% RSLogix 500 project Blue Banner Dump Line SLC 500.RSS, saved by version 11.00.00.00 %
PROJECT "BLUEBANR"    % processor: type code 8 %

PROGRAM FILES
  LAD 2   56 rungs

DATA FILES
  O0 OUTPUT  2 elements
  I1 INPUT  3 elements
  S2 STATUS  16 elements
  B3 BINARY  3 elements
  T4 TIMER  18 elements
  C5 COUNTER  1 elements
  R6 CONTROL  1 elements
  N7 INTEGER  1 elements

LADDER 2
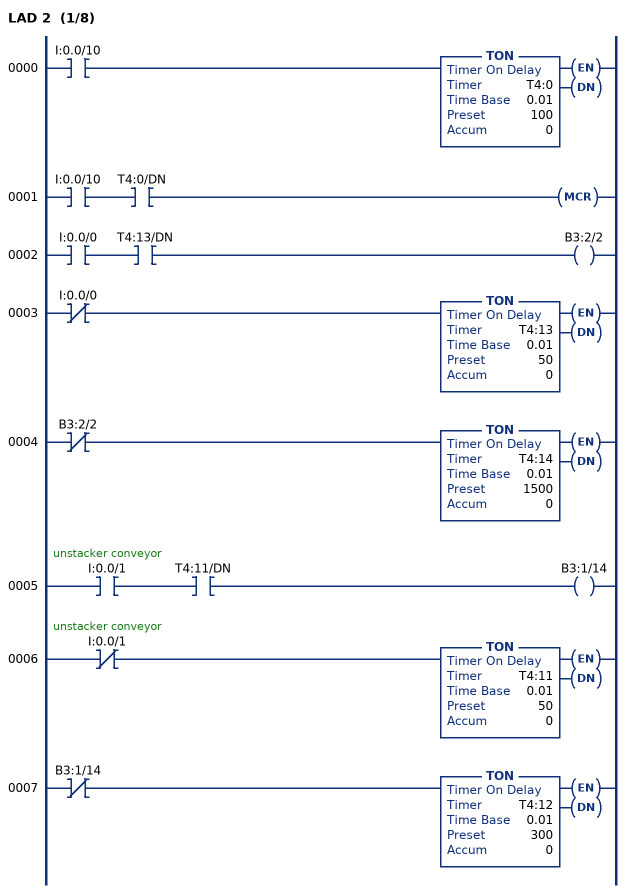
% Rung: 0 %
SOR XIC I:0.0/10 TON T4:0 0.01 100 0 EOR
% Rung: 1 %
SOR XIC I:0.0/10 XIC T4:0/DN MCR EOR
% Rung: 2 %
SOR XIC I:0.0/0 XIC T4:13/DN OTE B3:2/2 EOR
% Rung: 3 %
SOR XIO I:0.0/0 TON T4:13 0.01 50 0 EOR
% Rung: 4 %
SOR XIO B3:2/2 TON T4:14 0.01 1500 0 EOR
% Rung: 5 %
SOR XIC I:0.0/1 XIC T4:11/DN OTE B3:1/14 EOR
%   I:0.0/1  "unstacker conveyor" %
% Rung: 6 %
SOR XIO I:0.0/1 TON T4:11 0.01 50 0 EOR
%   I:0.0/1  "unstacker conveyor" %
% Rung: 7 %
SOR XIO B3:1/14 TON T4:12 0.01 300 0 EOR

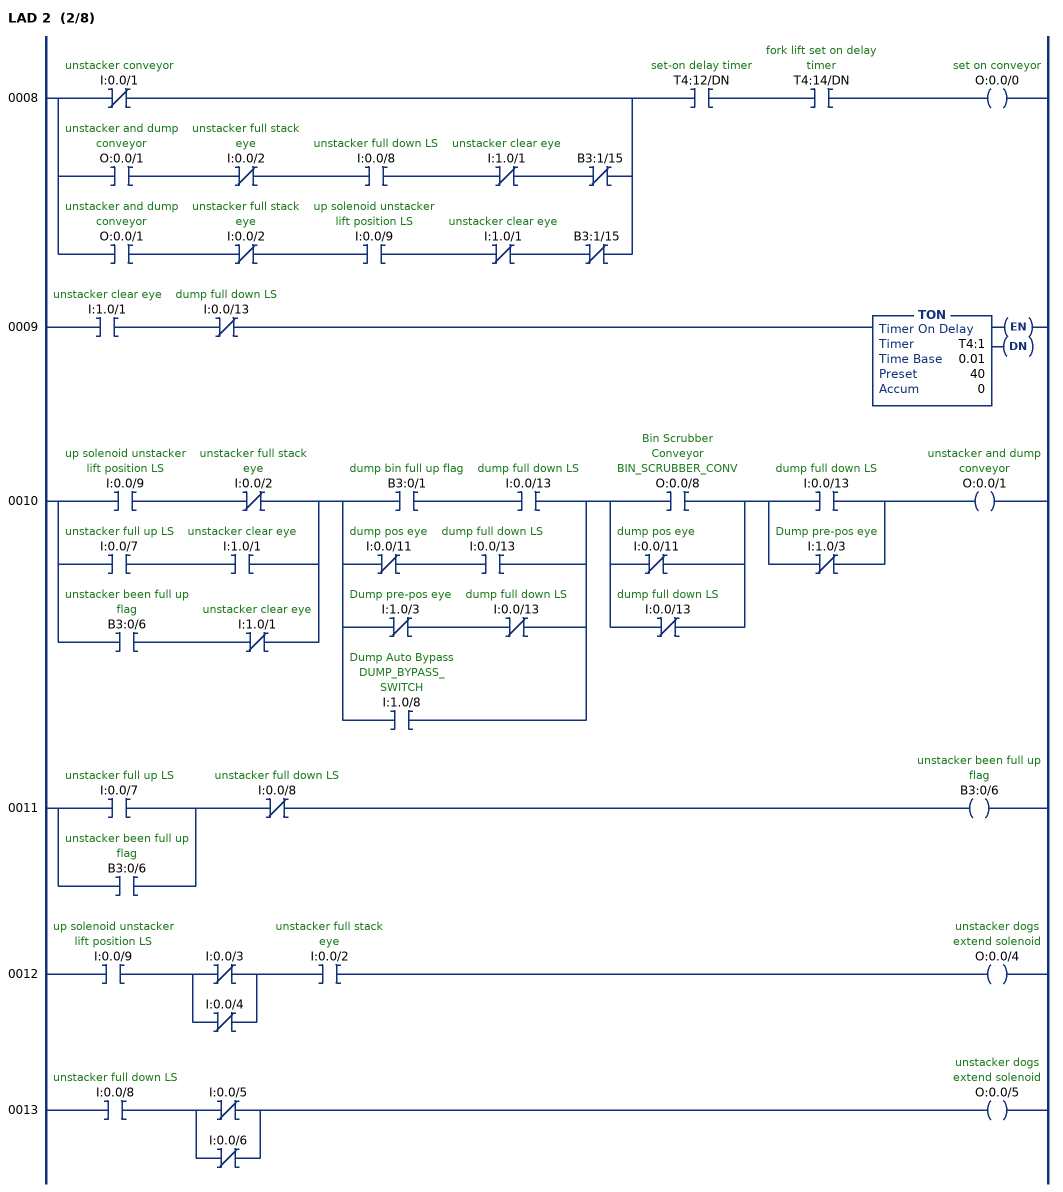
% Rung: 8 %
SOR BST XIO I:0.0/1 NXB XIC O:0.0/1 XIO I:0.0/2 XIC I:0.0/8 XIO I:1.0/1 XIO B3:1/15 NXB XIC O:0.0/1 XIO I:0.0/2 XIC I:0.0/9 XIO I:1.0/1 XIO B3:1/15 BND XIC T4:12/DN XIC T4:14/DN OTE O:0.0/0 EOR
%   I:0.0/1  "unstacker conveyor" %
%   O:0.0/1  "unstacker and dump conveyor" %
%   I:0.0/2  "unstacker full stack eye" %
%   I:0.0/8  "unstacker full down LS" %
%   I:1.0/1  "unstacker clear eye" %
%   I:0.0/9  "up solenoid unstacker lift position LS" %
%   T4:12/DN  "set-on delay timer" %
%   T4:14/DN  "fork lift set on delay timer" %
%   O:0.0/0  "set on conveyor" %
% Rung: 9 %
SOR XIC I:1.0/1 XIO I:0.0/13 TON T4:1 0.01 40 0 EOR
%   I:1.0/1  "unstacker clear eye" %
%   I:0.0/13  "dump full down LS" %
% Rung: 10 %
SOR BST XIC I:0.0/9 XIO I:0.0/2 NXB XIC I:0.0/7 XIC I:1.0/1 NXB XIC B3:0/6 XIO I:1.0/1 BND BST XIC B3:0/1 XIC I:0.0/13 NXB XIO I:0.0/11 XIC I:0.0/13 NXB BST XIO I:1.0/3 XIO I:0.0/13 NXB XIC I:1.0/8 BND BND BST XIC O:0.0/8 NXB XIO I:0.0/11 NXB XIO I:0.0/13 BND BST XIC I:0.0/13 NXB XIO I:1.0/3 BND OTE O:0.0/1 EOR
%   I:0.0/9  "up solenoid unstacker lift position LS" %
%   I:0.0/2  "unstacker full stack eye" %
%   I:0.0/7  "unstacker full up LS" %
%   I:1.0/1  "unstacker clear eye" %
%   B3:0/6  "unstacker been full up flag" %
%   B3:0/1  "dump bin full up flag" %
%   I:0.0/13  "dump full down LS" %
%   I:0.0/11  "dump pos eye" %
%   I:1.0/3  "Dump pre-pos eye" %
%   I:1.0/8  DUMP_BYPASS_SWITCH  "Dump Auto Bypass" %
%   O:0.0/8  BIN_SCRUBBER_CONV  "Bin Scrubber Conveyor" %
%   O:0.0/1  "unstacker and dump conveyor" %
% Rung: 11 %
SOR BST XIC I:0.0/7 NXB XIC B3:0/6 BND XIO I:0.0/8 OTE B3:0/6 EOR
%   I:0.0/7  "unstacker full up LS" %
%   B3:0/6  "unstacker been full up flag" %
%   I:0.0/8  "unstacker full down LS" %
% Rung: 12 %
SOR XIC I:0.0/9 BST XIO I:0.0/3 NXB XIO I:0.0/4 BND XIC I:0.0/2 OTE O:0.0/4 EOR
%   I:0.0/9  "up solenoid unstacker lift position LS" %
%   I:0.0/2  "unstacker full stack eye" %
%   O:0.0/4  "unstacker dogs extend solenoid" %
% Rung: 13 %
SOR XIC I:0.0/8 BST XIO I:0.0/5 NXB XIO I:0.0/6 BND OTE O:0.0/5 EOR
%   I:0.0/8  "unstacker full down LS" %
%   O:0.0/5  "unstacker dogs extend solenoid" %

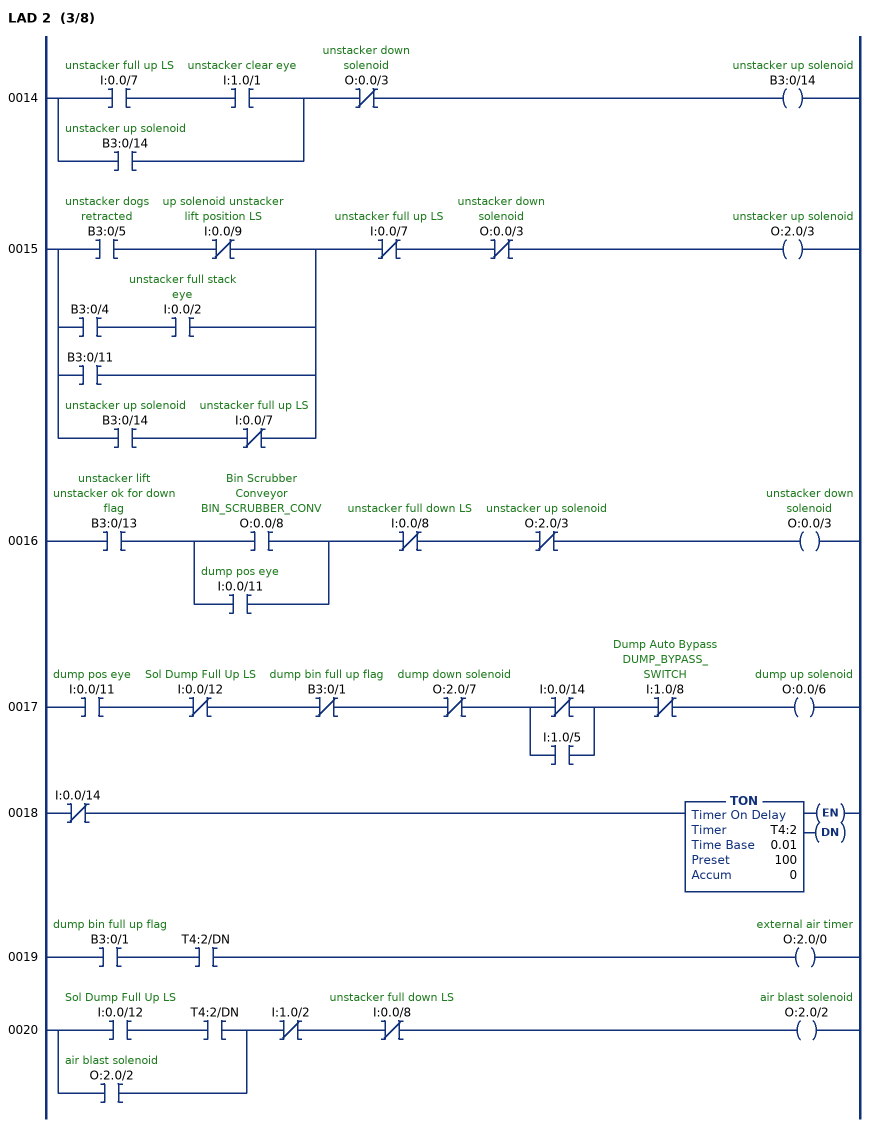
% Rung: 14 %
SOR BST XIC I:0.0/7 XIC I:1.0/1 NXB XIC B3:0/14 BND XIO O:0.0/3 OTE B3:0/14 EOR
%   I:0.0/7  "unstacker full up LS" %
%   I:1.0/1  "unstacker clear eye" %
%   B3:0/14  "unstacker up solenoid" %
%   O:0.0/3  "unstacker down solenoid" %
% Rung: 15 %
SOR BST XIC B3:0/5 XIO I:0.0/9 NXB XIC B3:0/4 XIC I:0.0/2 NXB XIC B3:0/11 NXB XIC B3:0/14 XIO I:0.0/7 BND XIO I:0.0/7 XIO O:0.0/3 OTE O:2.0/3 EOR
%   B3:0/5  "unstacker dogs retracted" %
%   I:0.0/9  "up solenoid unstacker lift position LS" %
%   I:0.0/2  "unstacker full stack eye" %
%   B3:0/14  "unstacker up solenoid" %
%   I:0.0/7  "unstacker full up LS" %
%   O:0.0/3  "unstacker down solenoid" %
%   O:2.0/3  "unstacker up solenoid" %
% Rung: 16 %
SOR XIC B3:0/13 BST XIC O:0.0/8 NXB XIC I:0.0/11 BND XIO I:0.0/8 XIO O:2.0/3 OTE O:0.0/3 EOR
%   B3:0/13  "unstacker lift unstacker ok for down flag" %
%   O:0.0/8  BIN_SCRUBBER_CONV  "Bin Scrubber Conveyor" %
%   I:0.0/11  "dump pos eye" %
%   I:0.0/8  "unstacker full down LS" %
%   O:2.0/3  "unstacker up solenoid" %
%   O:0.0/3  "unstacker down solenoid" %
% Rung: 17 %
SOR XIC I:0.0/11 XIO I:0.0/12 XIO B3:0/1 XIO O:2.0/7 BST XIO I:0.0/14 NXB XIC I:1.0/5 BND XIO I:1.0/8 OTE O:0.0/6 EOR
%   I:0.0/11  "dump pos eye" %
%   I:0.0/12  "Sol Dump Full Up LS" %
%   B3:0/1  "dump bin full up flag" %
%   O:2.0/7  "dump down solenoid" %
%   I:1.0/8  DUMP_BYPASS_SWITCH  "Dump Auto Bypass" %
%   O:0.0/6  "dump up solenoid" %
% Rung: 18 %
SOR XIO I:0.0/14 TON T4:2 0.01 100 0 EOR
% Rung: 19 %
SOR XIC B3:0/1 XIC T4:2/DN OTE O:2.0/0 EOR
%   B3:0/1  "dump bin full up flag" %
%   O:2.0/0  "external air timer" %
% Rung: 20 %
SOR BST XIC I:0.0/12 XIC T4:2/DN NXB XIC O:2.0/2 BND XIO I:1.0/2 XIO I:0.0/8 OTE O:2.0/2 EOR
%   I:0.0/12  "Sol Dump Full Up LS" %
%   O:2.0/2  "air blast solenoid" %
%   I:0.0/8  "unstacker full down LS" %

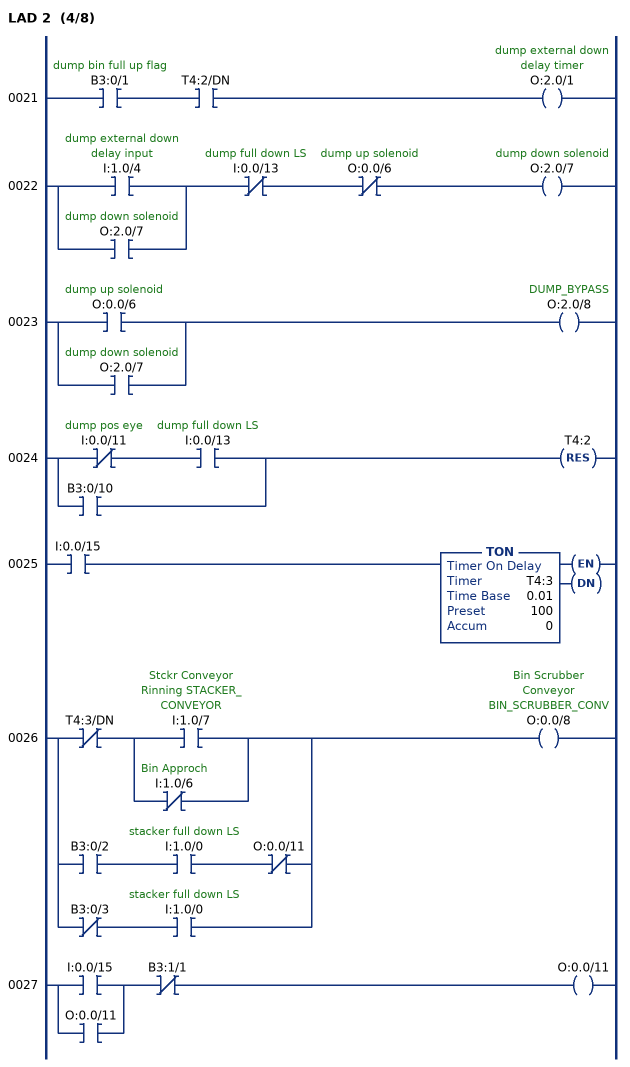
% Rung: 21 %
SOR XIC B3:0/1 XIC T4:2/DN OTE O:2.0/1 EOR
%   B3:0/1  "dump bin full up flag" %
%   O:2.0/1  "dump external down delay timer" %
% Rung: 22 %
SOR BST XIC I:1.0/4 NXB XIC O:2.0/7 BND XIO I:0.0/13 XIO O:0.0/6 OTE O:2.0/7 EOR
%   I:1.0/4  "dump external down delay input" %
%   O:2.0/7  "dump down solenoid" %
%   I:0.0/13  "dump full down LS" %
%   O:0.0/6  "dump up solenoid" %
% Rung: 23 %
SOR BST XIC O:0.0/6 NXB XIC O:2.0/7 BND OTE O:2.0/8 EOR
%   O:0.0/6  "dump up solenoid" %
%   O:2.0/7  "dump down solenoid" %
%   O:2.0/8  DUMP_BYPASS %
% Rung: 24 %
SOR BST XIO I:0.0/11 XIC I:0.0/13 NXB XIC B3:0/10 BND RES T4:2 EOR
%   I:0.0/11  "dump pos eye" %
%   I:0.0/13  "dump full down LS" %
% Rung: 25 %
SOR XIC I:0.0/15 TON T4:3 0.01 100 0 EOR
% Rung: 26 %
SOR BST XIO T4:3/DN BST XIC I:1.0/7 NXB XIO I:1.0/6 BND NXB XIC B3:0/2 XIC I:1.0/0 XIO O:0.0/11 NXB XIO B3:0/3 XIC I:1.0/0 BND OTE O:0.0/8 EOR
%   I:1.0/7  STACKER_CONVEYOR  "Stckr Conveyor Rinning" %
%   I:1.0/6  "Bin Approch" %
%   I:1.0/0  "stacker full down LS" %
%   O:0.0/8  BIN_SCRUBBER_CONV  "Bin Scrubber Conveyor" %
% Rung: 27 %
SOR BST XIC I:0.0/15 NXB XIC O:0.0/11 BND XIO B3:1/1 OTE O:0.0/11 EOR

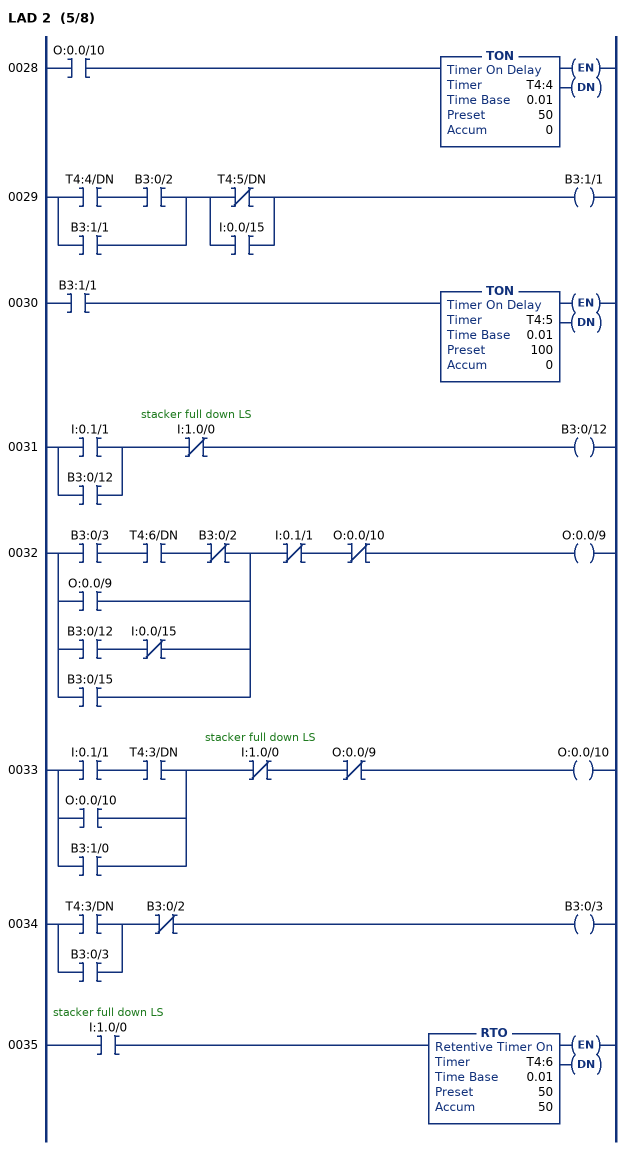
% Rung: 28 %
SOR XIC O:0.0/10 TON T4:4 0.01 50 0 EOR
% Rung: 29 %
SOR BST XIC T4:4/DN XIC B3:0/2 NXB XIC B3:1/1 BND BST XIO T4:5/DN NXB XIC I:0.0/15 BND OTE B3:1/1 EOR
% Rung: 30 %
SOR XIC B3:1/1 TON T4:5 0.01 100 0 EOR
% Rung: 31 %
SOR BST XIC I:0.1/1 NXB XIC B3:0/12 BND XIO I:1.0/0 OTE B3:0/12 EOR
%   I:1.0/0  "stacker full down LS" %
% Rung: 32 %
SOR BST XIC B3:0/3 XIC T4:6/DN XIO B3:0/2 NXB XIC O:0.0/9 NXB XIC B3:0/12 XIO I:0.0/15 NXB XIC B3:0/15 BND XIO I:0.1/1 XIO O:0.0/10 OTE O:0.0/9 EOR
% Rung: 33 %
SOR BST XIC I:0.1/1 XIC T4:3/DN NXB XIC O:0.0/10 NXB XIC B3:1/0 BND XIO I:1.0/0 XIO O:0.0/9 OTE O:0.0/10 EOR
%   I:1.0/0  "stacker full down LS" %
% Rung: 34 %
SOR BST XIC T4:3/DN NXB XIC B3:0/3 BND XIO B3:0/2 OTE B3:0/3 EOR
% Rung: 35 %
SOR XIC I:1.0/0 RTO T4:6 0.01 50 50 EOR
%   I:1.0/0  "stacker full down LS" %

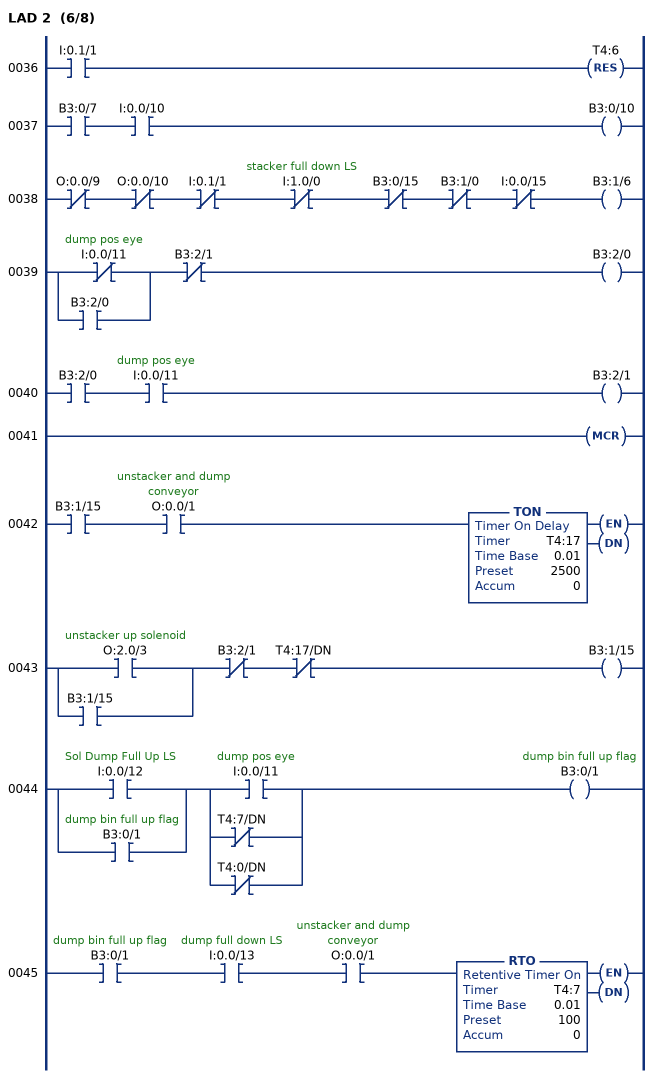
% Rung: 36 %
SOR XIC I:0.1/1 RES T4:6 EOR
% Rung: 37 %
SOR XIC B3:0/7 XIC I:0.0/10 OTE B3:0/10 EOR
% Rung: 38 %
SOR XIO O:0.0/9 XIO O:0.0/10 XIO I:0.1/1 XIO I:1.0/0 XIO B3:0/15 XIO B3:1/0 XIO I:0.0/15 OTE B3:1/6 EOR
%   I:1.0/0  "stacker full down LS" %
% Rung: 39 %
SOR BST XIO I:0.0/11 NXB XIC B3:2/0 BND XIO B3:2/1 OTE B3:2/0 EOR
%   I:0.0/11  "dump pos eye" %
% Rung: 40 %
SOR XIC B3:2/0 XIC I:0.0/11 OTE B3:2/1 EOR
%   I:0.0/11  "dump pos eye" %
% Rung: 41 %
SOR MCR EOR
% Rung: 42 %
SOR XIC B3:1/15 XIC O:0.0/1 TON T4:17 0.01 2500 0 EOR
%   O:0.0/1  "unstacker and dump conveyor" %
% Rung: 43 %
SOR BST XIC O:2.0/3 NXB XIC B3:1/15 BND XIO B3:2/1 XIO T4:17/DN OTE B3:1/15 EOR
%   O:2.0/3  "unstacker up solenoid" %
% Rung: 44 %
SOR BST XIC I:0.0/12 NXB XIC B3:0/1 BND BST XIC I:0.0/11 NXB XIO T4:7/DN NXB XIO T4:0/DN BND OTE B3:0/1 EOR
%   I:0.0/12  "Sol Dump Full Up LS" %
%   B3:0/1  "dump bin full up flag" %
%   I:0.0/11  "dump pos eye" %
% Rung: 45 %
SOR XIC B3:0/1 XIC I:0.0/13 XIC O:0.0/1 RTO T4:7 0.01 100 0 EOR
%   B3:0/1  "dump bin full up flag" %
%   I:0.0/13  "dump full down LS" %
%   O:0.0/1  "unstacker and dump conveyor" %

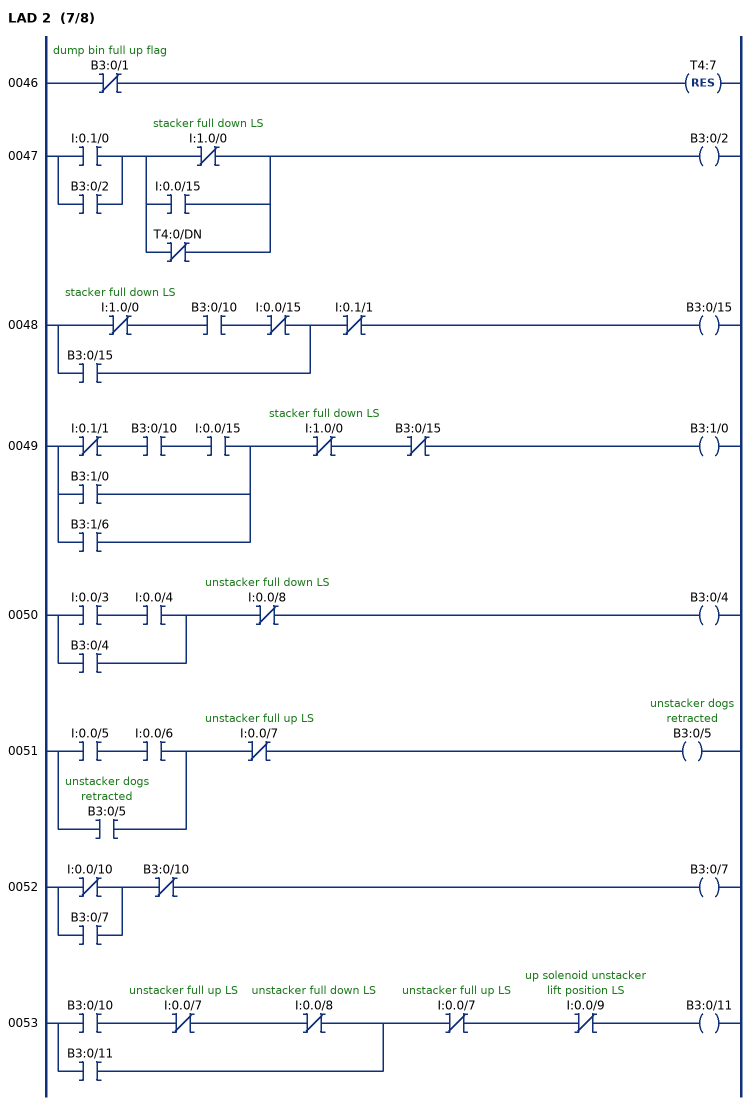
% Rung: 46 %
SOR XIO B3:0/1 RES T4:7 EOR
%   B3:0/1  "dump bin full up flag" %
% Rung: 47 %
SOR BST XIC I:0.1/0 NXB XIC B3:0/2 BND BST XIO I:1.0/0 NXB XIC I:0.0/15 NXB XIO T4:0/DN BND OTE B3:0/2 EOR
%   I:1.0/0  "stacker full down LS" %
% Rung: 48 %
SOR BST XIO I:1.0/0 XIC B3:0/10 XIO I:0.0/15 NXB XIC B3:0/15 BND XIO I:0.1/1 OTE B3:0/15 EOR
%   I:1.0/0  "stacker full down LS" %
% Rung: 49 %
SOR BST XIO I:0.1/1 XIC B3:0/10 XIC I:0.0/15 NXB XIC B3:1/0 NXB XIC B3:1/6 BND XIO I:1.0/0 XIO B3:0/15 OTE B3:1/0 EOR
%   I:1.0/0  "stacker full down LS" %
% Rung: 50 %
SOR BST XIC I:0.0/3 XIC I:0.0/4 NXB XIC B3:0/4 BND XIO I:0.0/8 OTE B3:0/4 EOR
%   I:0.0/8  "unstacker full down LS" %
% Rung: 51 %
SOR BST XIC I:0.0/5 XIC I:0.0/6 NXB XIC B3:0/5 BND XIO I:0.0/7 OTE B3:0/5 EOR
%   B3:0/5  "unstacker dogs retracted" %
%   I:0.0/7  "unstacker full up LS" %
% Rung: 52 %
SOR BST XIO I:0.0/10 NXB XIC B3:0/7 BND XIO B3:0/10 OTE B3:0/7 EOR
% Rung: 53 %
SOR BST XIC B3:0/10 XIO I:0.0/7 XIO I:0.0/8 NXB XIC B3:0/11 BND XIO I:0.0/7 XIO I:0.0/9 OTE B3:0/11 EOR
%   I:0.0/7  "unstacker full up LS" %
%   I:0.0/8  "unstacker full down LS" %
%   I:0.0/9  "up solenoid unstacker lift position LS" %

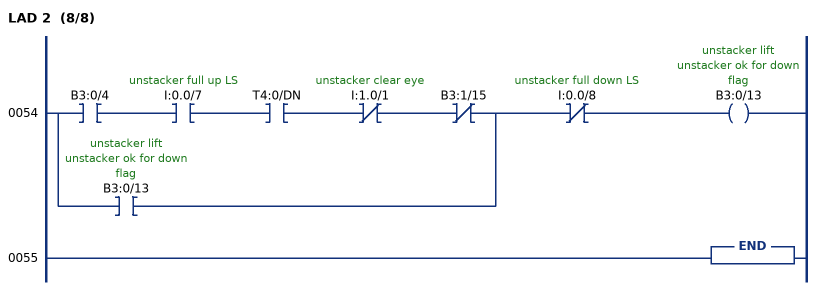
% Rung: 54 %
SOR BST XIC B3:0/4 XIC I:0.0/7 XIC T4:0/DN XIO I:1.0/1 XIO B3:1/15 NXB XIC B3:0/13 BND XIO I:0.0/8 OTE B3:0/13 EOR
%   I:0.0/7  "unstacker full up LS" %
%   I:1.0/1  "unstacker clear eye" %
%   B3:0/13  "unstacker lift unstacker ok for down flag" %
%   I:0.0/8  "unstacker full down LS" %
% Rung: 55 %
SOR END EOR

REVISION NOTES
  0: bbanner
  1: bban
  2: bb
  3: b
  4: bb
  5: bbb
  6: bbb
  7: Labels1
  8: labels2
  9: 4/6/2017

DATA TABLE (non-zero values as saved)
DATA B3
% B3:0 % 0XA090 0X0000 0X0000
DATA T4
% .PRE .ACC %
% T4:0 % 100 0
% T4:1 % 40 0
% T4:2 % 100 0
% T4:3 % 100 0
% T4:4 % 50 0
% T4:5 % 100 0
% T4:6 % 50 50
% T4:7 % 100 0
% T4:8 % 100 0
% T4:10 % 2500 0
% T4:11 % 50 0
% T4:12 % 300 0
% T4:13 % 50 0
% T4:14 % 1500 0
% T4:17 % 2500 0
